// TIA Portal project "CalcOnSCADA_05" (V14)

(* hardware
DEVICE "S71500/ET200MP station_1"  S7-1500 station
   slot 0: "Rail_0"  Rack  6ES7 590-1***0-0AA0
   slot 1: "PLC_1"  CPU 1513-1 PN  6ES7 513-1AL01-0AB0  V2.1
      slot 3: "CPU display_1"  6ES7591-1AA00-0AA0
DEVICE "HMI_1"  TP900 Comfort
   slot 0: "TP900 Comfort"  TP900 Comfort  6AV2 124-0JC01-0AX0  14.0.1.0
   slot 1: "HMI_RT_1"  TP900 Comfort  6AV2 124-0JC01-0AX0  14.0.1.0
   slot 5: "HMI_1.IE_CP_1"  PROFINET Interface  14.0.1.0
      slot 1: "PROFINET Interface_1"  PROFINET Interface
         slot 1: "Port_1"  Port
         slot 2: "Port_2"  Port
   slot 7: "HMI_1.MPI/DP_CP_1"  MPI/DP Interface  14.0.1.0
*)

// ===== PLC "PLC_1"  CPU 1513-1 PN =====

VAR_GLOBAL   // PLC tag table "Default tag table"
   "positive" AT %M515.0 : Bool;
   "positiveOut" AT %M515.1 : Bool;
END_VAR

VAR_GLOBAL   // PLC tag table "Tag table_1"
   "Watchable" AT %M100.0 : LReal;
   "hjbhb" AT %M108.0 : LReal;
   "mb514" AT %MB514 : Byte;
END_VAR

TYPE "Digit"
   STRUCT
      visiComa : Bool;
      visiMinus : Bool;
      visible2 : Bool;
      visible3 : Bool;
      visible4 : Bool;
      visible5 : Bool;
      visible6 : Bool;
      visible7 : Bool;
      visible8 : Bool;
      visible9 : Bool;
      visible10 : Bool;
      visible11 : Bool;
      visible12 : Bool;
      visible13 : Bool;
      visible14 : Bool;
      visible15 : Bool;
      digit : Word;
   END_STRUCT;
END_TYPE

TYPE "Button"
   STRUCT
      b00 : Bool;
      b01 : Bool;
      b02 : Bool;
      b03 : Bool;
      b04 : Bool;
      b05 : Bool;
      click : Bool;
      oldClick : Bool;
   END_STRUCT;
END_TYPE

TYPE "Number"
   STRUCT
      coma : Bool;
      initOk : Bool;
      num2 : Bool;
      num3 : Bool;
      num4 : Bool;
      num5 : Bool;
      num6 : Bool;
      num7 : Bool;
      longI : LInt;
      I : Int;
      longTr : LReal;
      Tr : Real;
      longR : LReal;
      R : Real;
      pos : Int;   // Кількість десяткових розрядів
      posC : Int;   // Позиція коми
      posR : LInt;   // Вага десяткового розряду
   END_STRUCT;
END_TYPE

DATA_BLOCK "NUMs"   // DB1
{ S7_Optimized_Access := 'TRUE' }
VERSION : 0.1
   VAR
      Num : Array[0..31] of "Number";
      TEMP : Array[0..17] of LReal;
      TEMP2 : Array[0..17] of LInt;
      FaceLongI : String;
      FaceI : String;
      FaceLongR : String;
      FaceR : String;
      Index : Int;   // Індекс у масиві Num
      Action : Int;
      ActionBit : Bool;
      ActBit : Bool;   // Щоб виконати дію без =
      EquaBit : Bool;
      FaceLongFr : String;
      FaceFr : String;
      SizeI : Int;
      SizeAll : Int;
      Error : Bool;
      preError : Bool;
      TEN : Array[0..15] of LReal;
      bTEN : Array[0..15] of LReal;
   END_VAR
BEGIN
   bTEN[0] := 1.0E-15;
   bTEN[1] := 1.0E-14;
   bTEN[2] := 1.0E-13;
   bTEN[3] := 1.0E-12;
   bTEN[15] := 1.0;
   bTEN[9] := 1.0E-06;
   bTEN[10] := 1.0E-05;
   bTEN[11] := 0.0001;
   bTEN[12] := 0.001;
   bTEN[13] := 0.01;
   bTEN[14] := 0.1;
   bTEN[4] := 1.0E-11;
   bTEN[5] := 1.0E-10;
   bTEN[6] := 1.0E-09;
   bTEN[7] := 1.0E-08;
   bTEN[8] := 1.0E-07;
   TEN[0] := 1.0;
   TEN[1] := 10.0;
   TEN[2] := 100.0;
   TEN[3] := 1000.0;
   TEN[4] := 10000.0;
   TEN[5] := 100000.0;
   TEN[6] := 1000000.0;
   TEN[7] := 10000000.0;
   TEN[8] := 100000000.0;
   TEN[9] := 1000000000.0;
   TEN[10] := 10000000000.0;
   TEN[11] := 100000000000.0;
   TEN[12] := 1000000000000.0;
   TEN[13] := 10000000000000.0;
   TEN[14] := 100000000000000.0;
   TEN[15] := 1.0E+15;
END_DATA_BLOCK

// folder: Group_Misc

DATA_BLOCK "Digit_bl_10"   // DB10
{ S7_Optimized_Access := 'TRUE' }
VERSION : 0.1
   VAR
      Header : ArrayDBHeader;
      THIS : Array[0..15] of "Digit";
   END_VAR
BEGIN
   Header.LowerBound := 0;
   Header.UpperBound := 15;
   Header.Elements := 16;
   Header.PaddedSize := 18;
   Header.ElementSize := 18;
   THIS[0].digit := 16#1;
END_DATA_BLOCK

DATA_BLOCK "Butt_bl_200"   // DB200
{ S7_Optimized_Access := 'TRUE' }
VERSION : 0.1
   VAR
      Header : ArrayDBHeader;
      THIS : Array[0..31] of "Button";
   END_VAR
BEGIN
   Header.LowerBound := 0;
   Header.UpperBound := 31;
   Header.Elements := 32;
   Header.PaddedSize := 8;
   Header.ElementSize := 8;
END_DATA_BLOCK

// folder: System blocks/Program resources

DATA_BLOCK "DB_Timer_0"   // DB2
{ S7_Optimized_Access := 'TRUE' }
AUTHOR : Simatic
FAMILY : IEC
NAME : IEC_TMR
VERSION : 1.0
// stored: InstanceOfName IEC_TIMER
"IEC_TIMER"
BEGIN
END_DATA_BLOCK

// folder: (top level)

FUNCTION "Block_NumToD" : Void   // FC15, SCL
{ S7_Optimized_Access := 'TRUE' }
VERSION : 0.1
   VAR_INPUT
      inNumber : "Number";
   END_VAR
   VAR_TEMP
      tFaceLongR : String;
      tFaceLongI : String;
      tSizeAll : Int;
      tSizeFr : Int;
      ii : Int;
      i2 : Int;
      tShift : Word;
      tInt : Int;
      tShortStr : String;
      tDLongR : LReal;
      tLongR : LReal;
      tLongR2 : LReal;
      tLongI : LInt;
      tLongTr : LReal;
   END_VAR
   VAR CONSTANT
      word1 : Word := 16#1;
   END_VAR
BEGIN

   (*IF #inNumber.longI < 0 THEN
       #tAbsLongI := - #inNumber.longI; //знаходимо модуль
   ELSE
       #tAbsLongI := #inNumber.longI; //знаходимо модуль
   END_IF;
   #tAbsLongI := ABS(#inNumber.longI);*)

   #tFaceLongI      := S_CONV(#inNumber.longI);
   //"NUMs".FaceLongI := #tFaceLongI;
   "NUMs".FaceI     := S_CONV(#inNumber.I);
   #tFaceLongR      := S_CONV(#inNumber.longR);
   "NUMs".FaceLongR := #tFaceLongR;
   "NUMs".FaceR     := S_CONV(#inNumber.R);
   //"NUMs".FaceR := FC30(#tNumber.R);
   //"NUMs".FaceLongFr:= LREAL_TO_STRING(#inNumber.longTr);
   //"NUMs".FaceFr    := REAL_TO_STRING(#inNumber.Tr);

   #tLongR := ABS(#inNumber.longR);
   //#tLongR := ABS(#tLongR);
   #tLongI := ABS(#inNumber.longI);
   //#tLongI := ABS(#tLongI);
   #tLongTr := ABS(#inNumber.longTr);
   #tDLongR := #tLongR - #tLongTr;
   (*#tLongR := #inNumber.longR;
   #tLongI := #inNumber.longI;
   #tLongR := #tLongR * 10;
   #tLongI := LREAL_TO_LINT(#tLongR - 0.4999);
   #tDLongR := #tLongR - #tLongI;*)
   (*#i2 := 100;
   WHILE #ii <5 AND #i2 < 110 DO
       #ii += 1;
       #i2 += 1;
   END_WHILE;*)
   "NUMs".SizeI := LEN(#tFaceLongI); //намагаємося вирахувати кількість знакомісць до коми
   IF #tLongI < 1 THEN
       "NUMs".SizeI := 1;
   ELSE
       "NUMs".SizeI -= 1;
   END_IF;
   //"NUMs".TEMP[1]:=0;
   #tSizeFr := 0;    // 123456789012345
   WHILE #tDLongR > "NUMs".bTEN[#tSizeFr] AND #tSizeFr < (16-"NUMs".SizeI) DO
       "NUMs".TEMP[#tSizeFr] := #tDLongR;
       #tSizeFr += 1;
       //#tLongR := #tLongR * 10;
       #tLongR2 := "NUMs".TEN[#tSizeFr] * #tLongR ;
       //"NUMs".TEN[#tSizeFr] += 1;
       #tLongI := TRUNC(#tLongR2);
       "NUMs".TEMP2[#tSizeFr-1] := #tLongI;
       //#tInt := LREAL_TO_INT(#tLongR2 - 0.5);
       #tDLongR := #tLongR2 - LINT_TO_LREAL(#tLongI);  // +0.0000000000001;
       //#tDLongR := #tLongR2 - #tInt;
   END_WHILE;
   "NUMs".TEMP[#tSizeFr] := 88888888888888;
   "NUMs".TEMP2[#tSizeFr] := 88888888888888;

   #tFaceLongI := S_CONV(#tLongI);
   "NUMs".FaceLongI := #tFaceLongI;

   #tSizeAll := LEN(#tFaceLongI);
   "NUMs".SizeAll := #tSizeAll;
   "Block_CLS"();
   #tSizeAll := #tSizeAll - 1;
   (*
   #tShortStr := MID(IN := #tFaceLongI, L := 1, P := 2);
   #tInt := STRING_TO_INT(#tShortStr);
   #tShift := SHL(IN := #word1, N := #tInt);
   "Digit_bl_10"."THIS"[0].digit := #tShift;
   *)
   FOR #ii := 1 TO #tSizeAll DO
       #tShift := SHL(IN := #word1, N := S_CONV(MID(IN := #tFaceLongI, L := 1, P := #ii + 1)));
       "Digit_bl_10".THIS[#tSizeAll - #ii].digit := #tShift;
   END_FOR;
   IF #tSizeFr > 0 THEN
       "Digit_bl_10".THIS[#tSizeFr].visiComa := TRUE;
   END_IF;

   #ii := #tSizeFr;
   IF #tSizeAll>#tSizeFr THEN
       #inNumber.pos := #tSizeAll - 1;     //задля "Block_setMinus"
   ELSE
       #inNumber.pos := #tSizeFr;     //задля "Block_setMinus"
       REPEAT
           "Digit_bl_10".THIS[#ii].digit := 1;
           #ii -= 1;
       UNTIL (#ii-#tSizeAll)<0
       END_REPEAT;
   END_IF;

   "Block_setMinus"();
END_FUNCTION

FUNCTION "Block_100" : Void   // FC100, SCL
{ S7_Optimized_Access := 'TRUE' }
VERSION : 0.1
   VAR_TEMP
      ii : Int;
      tpos : Int;
      tButton : "Button";
      tLReal : LReal;
      tLInt : LInt;
   END_VAR
BEGIN


   //      =
   #tButton := "Butt_bl_200".THIS[24];
   IF (#tButton.click <> #tButton.oldClick) AND NOT "NUMs".Error THEN
       "Block_Equal"();
   END_IF;
   //      /
   #tButton := "Butt_bl_200".THIS[20];
   IF #tButton.click <> #tButton.oldClick THEN
       "Block_Action"();
       "NUMs".Action := 4;
   END_IF;
   //      *
   #tButton := "Butt_bl_200".THIS[21];
   IF #tButton.click <> #tButton.oldClick THEN
       "Block_Action"();
       "NUMs".Action := 3;
   END_IF;
   //      -
   #tButton := "Butt_bl_200".THIS[22];
   IF #tButton.click <> #tButton.oldClick THEN
       "Block_Action"();
       "NUMs".Action := 2;
   END_IF;
   //      +
   #tButton := "Butt_bl_200".THIS[23];
   IF #tButton.click <> #tButton.oldClick THEN
       "Block_Action"();
       "NUMs".Action := 1;
   END_IF;

   //      Coma
   #tButton := "Butt_bl_200".THIS[12];
   IF #tButton.click <> #tButton.oldClick THEN
       "NUMs".Num["NUMs".Index].initOk := true;
       IF "NUMs".Num["NUMs".Index].coma THEN
           ;
       ELSE
           "Digit_bl_10".THIS[0].visiComa := true;
       END_IF;
       "NUMs".Num["NUMs".Index].coma := true;
   END_IF;
   //      CE
   #tButton := "Butt_bl_200".THIS[17];
   IF #tButton.click <> #tButton.oldClick THEN
       "Block_CE"();
   END_IF;
   //      C
   #tButton := "Butt_bl_200".THIS[18];
   IF #tButton.click <> #tButton.oldClick THEN
       "Block_C"();
   END_IF;
   //      0
   #tButton := "Butt_bl_200".THIS[10];
   IF #tButton.click <> #tButton.oldClick AND ("NUMs".Num["NUMs".Index].pos < 15) THEN
       "Block_num Butt" ( iInt:=0, iDigit:=1 );
   END_IF;
   //      1
   #tButton := "Butt_bl_200".THIS[1];
   IF #tButton.click <> #tButton.oldClick AND ("NUMs".Num["NUMs".Index].pos < 15) THEN
       "Block_num Butt" ( iInt:=1, iDigit:=2 );
   END_IF;
   //      2
   #tButton := "Butt_bl_200".THIS[2];
   IF #tButton.click <> #tButton.oldClick AND ("NUMs".Num["NUMs".Index].pos < 15) THEN
       "Block_num Butt" ( iInt:=2, iDigit:=4 );
   END_IF;
   //      3
   #tButton := "Butt_bl_200".THIS[3];
   IF #tButton.click <> #tButton.oldClick AND ("NUMs".Num["NUMs".Index].pos < 15) THEN
       "Block_num Butt" ( iInt:=3, iDigit:=8 );
   END_IF;
   //      4
   #tButton := "Butt_bl_200".THIS[4];
   IF #tButton.click <> #tButton.oldClick AND ("NUMs".Num["NUMs".Index].pos < 15) THEN
       "Block_num Butt"(iInt := 4, iDigit := 16);
   END_IF;
   //      5
   #tButton := "Butt_bl_200".THIS[5];
   IF #tButton.click <> #tButton.oldClick AND ("NUMs".Num["NUMs".Index].pos < 15) THEN
       "Block_num Butt" ( iInt:=5, iDigit:=32 );
   END_IF;
   //      6
   #tButton := "Butt_bl_200".THIS[6];
   IF #tButton.click <> #tButton.oldClick AND ("NUMs".Num["NUMs".Index].pos < 15) THEN
       "Block_num Butt" ( iInt:=6, iDigit:=64 );
   END_IF;
   //      7
   #tButton := "Butt_bl_200".THIS[7];
   IF #tButton.click <> #tButton.oldClick AND ("NUMs".Num["NUMs".Index].pos < 15) THEN
       "Block_num Butt" ( iInt:=7, iDigit:=128 );
   END_IF;
   //      8
   #tButton := "Butt_bl_200".THIS[8];
   IF #tButton.click <> #tButton.oldClick AND ("NUMs".Num["NUMs".Index].pos < 15) THEN
       "Block_num Butt"(iInt := 8, iDigit := 256);
   END_IF;
   //      9
   #tButton := "Butt_bl_200".THIS[9];
   IF #tButton.click <> #tButton.oldClick AND ("NUMs".Num["NUMs".Index].pos < 15) THEN
       "Block_num Butt" ( iInt:=9, iDigit:=512 );
   END_IF;

   //      +-
   #tButton := "Butt_bl_200".THIS[11];
   IF (#tButton.click <> #tButton.oldClick) AND NOT "NUMs".Error THEN
       "Block_Minus"();
   END_IF;
END_FUNCTION

ORGANIZATION_BLOCK "Main"   // OB1, STL, ProgramCycle
TITLE = "Main Program Sweep (Cycle)"
{ S7_Optimized_Access := 'TRUE' }
VERSION : 0.1
   VAR_INPUT
      Initial_Call : Bool;   // Initial call of this OB
      Remanence : Bool;   // =True, if remanent data are available
   END_VAR
BEGIN

REGION Network 1
         CALL  "Block_100";
END_REGION

REGION Network 2
         CALL  "Block_200";
END_REGION

REGION Network 3
         CALL  "Block_99";
END_REGION
END_ORGANIZATION_BLOCK

ORGANIZATION_BLOCK "Programming error"   // OB121, LAD, ProgrammingError
{ S7_Optimized_Access := 'TRUE' }
VERSION : 0.1
   VAR_INPUT
      BlockNr : UInt;   // Number of causing block
      Reaction : USInt;   // 0:ignore, 1:substitute, 2:skip
      Fault_ID : Byte;   // Fault identifier
      BlockType : USInt;   // 16#01:OB, 16#02:FC, 16#03:FB, 16#04:SFC, 16#05:SFB, 16#06:DB: Type of block causing the error
      Area : USInt;   // Area where the error occured
      DBNr : DB_ANY;   // DB number if Area = DB or DI
      Csg_OBNr : OB_Any;   // Number of OB causing the error
      Csg_Prio : USInt;   // Priority of OB causing the error
      Width : USInt;   // 0:bit, 1:byte, 2:word, 3:dword, 4:lword
   END_VAR
BEGIN

REGION Network 1
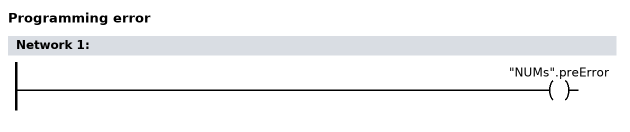
   RUNG wire#powerrail
      Coil( "NUMs".preError )
   END_RUNG
   // the same network as SCL:
   "NUMs".preError := TRUE;
END_REGION
END_ORGANIZATION_BLOCK

// folder: Group_100

FUNCTION "Block_CLS" : Void   // FC2, SCL
{ S7_Optimized_Access := 'TRUE' }
VERSION : 0.1
   VAR_TEMP
      ii : Int;
   END_VAR
BEGIN


   FOR #ii := 0 TO 15 DO
       "Digit_bl_10".THIS[#ii].digit := 0;
   END_FOR;
   "Block_unComa"();   //прибираю коми
   "Block_unMinus"();  //прибираю мінуси
END_FUNCTION

FUNCTION "Block_num Butt" : Void   // FC11, SCL
{ S7_Optimized_Access := 'TRUE' }
VERSION : 0.1
   VAR_INPUT
      iDigit : Word;
      iInt : Int;
   END_VAR
   VAR_TEMP
      tpos : Int;
      tLReal : LReal;
   END_VAR
BEGIN

   IF "NUMs".Error THEN
       "Block_C"();
   END_IF;

   IF "NUMs".ActionBit THEN
       "Block_CE"();
       "NUMs".ActionBit := false;
   END_IF;

   IF "NUMs".EquaBit THEN
       "Block_CE"();
       "NUMs".EquaBit := false;
   END_IF;

   IF "NUMs".Num["NUMs".Index].initOk THEN
       "NUMs".Num["NUMs".Index].pos += 1;
       #tpos := "NUMs".Num["NUMs".Index].pos;
       WHILE #tpos > 0 DO
           "Digit_bl_10".THIS[#tpos].digit :=
           "Digit_bl_10".THIS[#tpos - 1].digit;
           #tpos -= 1;
       END_WHILE;
       IF "NUMs".Num["NUMs".Index].coma THEN
           "NUMs".Num["NUMs".Index].posR *=10;
           #tLReal := #iInt;
           "NUMs".Num["NUMs".Index].longR :=
           #tLReal / "NUMs".Num["NUMs".Index].posR + "NUMs".Num["NUMs".Index].longR;
           "NUMs".Num["NUMs".Index].R := "NUMs".Num["NUMs".Index].longR;   //звичайний ріел
           (*        
           "NUMs".Num["NUMs".Index].longFr :=
           "NUMs".Num["NUMs".Index].longR - "NUMs".Num["NUMs".Index].longI;
           *)
           "NUMs".Num["NUMs".Index].longTr :=
           #tLReal / "NUMs".Num["NUMs".Index].posR + "NUMs".Num["NUMs".Index].longTr;
           "NUMs".Num["NUMs".Index].Tr := "NUMs".Num["NUMs".Index].longTr;
       ELSE
           "NUMs".Num["NUMs".Index].longI := 10 * "NUMs".Num["NUMs".Index].longI + #iInt;
           "NUMs".Num["NUMs".Index].I := 10 * "NUMs".Num["NUMs".Index].I + #iInt;
           "NUMs".Num["NUMs".Index].longR := 10 * "NUMs".Num["NUMs".Index].longR + #iInt;
           "NUMs".Num["NUMs".Index].R := "NUMs".Num["NUMs".Index].longR;   //звичайний ріел
       END_IF;
   ELSE
       "NUMs".Num["NUMs".Index].longI := #iInt;
       "NUMs".Num["NUMs".Index].I := #iInt;
       "NUMs".Num["NUMs".Index].longR := #iInt;
       "NUMs".Num["NUMs".Index].R := #iInt;
   END_IF;

   "Digit_bl_10".THIS[0].digit := #iDigit; //

   IF "NUMs".Num["NUMs".Index].coma THEN
       "NUMs".Num["NUMs".Index].posC +=1;
       "Block_unComa"();//прибираю коми
       "Digit_bl_10".THIS["NUMs".Num["NUMs".Index].posC].visiComa := true;   //
   END_IF;
   "Block_setMinus"();

   IF #iInt = 0 THEN
       ;
   ELSE
       "NUMs".Num["NUMs".Index].initOk := true;
   END_IF;
END_FUNCTION

FUNCTION "Block_Equal" : Void   // FC12, SCL
{ S7_Optimized_Access := 'TRUE' }
VERSION : 0.1
   VAR_TEMP
      tLReal : LReal;
      tButton : "Button";
      tLInt : LInt;
   END_VAR
BEGIN

       "NUMs".Index := 0;
       #tLReal := "NUMs".Num[0].longR;
       CASE "NUMs".Action OF
           1:
               "NUMs".Num[0].longR := #tLReal + "NUMs".Num[1].longR;
           2:
               "NUMs".Num[0].longR := #tLReal - "NUMs".Num[1].longR;
           3:
               "NUMs".Num[0].longR := #tLReal * "NUMs".Num[1].longR;
           4:
               "NUMs".Num[0].longR := #tLReal / "NUMs".Num[1].longR;
       END_CASE;

   "Block_ActCase"();
   "Block_NumToD"("NUMs".Num[0]);

   "NUMs".EquaBit := TRUE;
   "NUMs".ActBit := FALSE;
END_FUNCTION

FUNCTION "Block_unComa" : Void   // FC13, SCL
{ S7_Optimized_Access := 'TRUE' }
VERSION : 0.1
   VAR_TEMP
      ii : Int;
   END_VAR
BEGIN

   FOR #ii := 0 TO 15 DO
       "Digit_bl_10".THIS[#ii].visiComa := FALSE;
   END_FOR;
END_FUNCTION

FUNCTION "Block_CE" : Void   // FC14, SCL
{ S7_Optimized_Access := 'TRUE' }
VERSION : 0.1
   VAR_TEMP
      ii : Int;
   END_VAR
BEGIN

   "Block_NumCE"("NUMs".Index);
END_FUNCTION

FUNCTION "Block_Zeroing" : Void   // FC16, SCL
{ S7_Optimized_Access := 'TRUE' }
VERSION : 0.1
   VAR_INPUT
      iIndex : Int;
   END_VAR
BEGIN


   "NUMs".Num[#iIndex].longI := 0;
   "NUMs".Num[#iIndex].I := 0;
   "NUMs".Num[#iIndex].longR := 0.0;
   "NUMs".Num[#iIndex].R := 0.0;
   "NUMs".Num[#iIndex].longTr := 0.0;
   "NUMs".Num[#iIndex].Tr := 0.0;
END_FUNCTION

FUNCTION "Block_C" : Void   // FC17, SCL
{ S7_Optimized_Access := 'TRUE' }
VERSION : 0.1
BEGIN

   "NUMs".ActionBit := FALSE;
   "NUMs".ActBit := FALSE;
   "NUMs".Action := 0;
   "NUMs".Index := 0;
   "Block_NumCE"(0);
   "Block_NumCE"(1);

   "NUMs".Error := FALSE;
   "NUMs".preError := FALSE;
END_FUNCTION

FUNCTION "Block_NumCE" : Void   // FC18, SCL
{ S7_Optimized_Access := 'TRUE' }
VERSION : 0.1
   VAR_INPUT
      iIndex : Int;
   END_VAR
BEGIN

   "NUMs".Num[#iIndex].initOk := false;
   "NUMs".Num[#iIndex].coma := false;
   "NUMs".Num[#iIndex].pos := 0;
   "NUMs".Num[#iIndex].posC := 0;
   "NUMs".Num[#iIndex].posR := 1;

   "Block_Zeroing"(#iIndex);
   "Block_CLS"();

   //"Digit_bl_10"."THIS"[0].visible0 := false;
   "Digit_bl_10".THIS[0].digit := 1;
END_FUNCTION

FUNCTION "Block_LAD" : Void   // FC19, LAD
{ S7_Optimized_Access := 'TRUE' }
VERSION : 0.1
BEGIN
END_FUNCTION

FUNCTION "Block_Action" : Void   // FC20, SCL
{ S7_Optimized_Access := 'TRUE' }
VERSION : 0.1
BEGIN

   IF "NUMs".ActBit AND (NOT "NUMs".ActionBit) THEN
       "Block_Equal"();
   END_IF;
   "NUMs".ActBit := TRUE;

   "NUMs".Index := 1;
   "NUMs".ActionBit := TRUE;
END_FUNCTION

FUNCTION "Block_ActCase" : Void   // FC21, SCL
{ S7_Optimized_Access := 'TRUE' }
VERSION : 0.1
BEGIN

   "NUMs".Num[0].R := "NUMs".Num[0].longR;
   (*"NUMs".Num[0].longFr := FRAC_LREAL("NUMs".Num[0].longR);
   "NUMs".Num[0].Fr := "NUMs".Num[0].longFr;*)

   //"NUMs".Num[0].longI := LREAL_TO_LINT("NUMs".Num[0].longR - 0.499999);
   "NUMs".Num[0].longI := TRUNC("NUMs".Num[0].longR);
   "NUMs".Num[0].I     := TRUNC("NUMs".Num[0].longR);

   "NUMs".Num[0].longTr := TRUNC("NUMs".Num[0].longR);
   "NUMs".Num[0].Tr     := TRUNC("NUMs".Num[0].longR);
END_FUNCTION

FUNCTION "Block_setMinus" : Void   // FC22, SCL
{ S7_Optimized_Access := 'TRUE' }
VERSION : 0.1
BEGIN


   IF "NUMs".Num["NUMs".Index].longR < 0 THEN
       "Block_unMinus"();  //прибираю мінуси
       "Digit_bl_10".THIS["NUMs".Num["NUMs".Index].pos].visiMinus := TRUE;        //
   END_IF;
END_FUNCTION

FUNCTION "Block_unMinus" : Void   // FC23, SCL
{ S7_Optimized_Access := 'TRUE' }
VERSION : 0.1
   VAR_TEMP
      ii : Int;
   END_VAR
BEGIN

   FOR #ii := 0 TO 15 DO
       "Digit_bl_10".THIS[#ii].visiMinus := FALSE;
   END_FOR;
END_FUNCTION

FUNCTION "Block_Minus" : Void   // FC101, SCL
{ S7_Optimized_Access := 'TRUE' }
VERSION : 0.1
BEGIN

   //"mb514" := "mb514" + 1;
   //invert
   "Digit_bl_10".THIS["NUMs".Num["NUMs".Index].pos].visiMinus := NOT "Digit_bl_10".THIS["NUMs".Num["NUMs".Index].pos].visiMinus;
   "NUMs".Num["NUMs".Index].longR := -"NUMs".Num["NUMs".Index].longR;



   //
END_FUNCTION

// folder: Group_200

FUNCTION "Block_200" : Void   // FC200, FBD
{ S7_Optimized_Access := 'TRUE' }
VERSION : 0.1
BEGIN

REGION Network 1
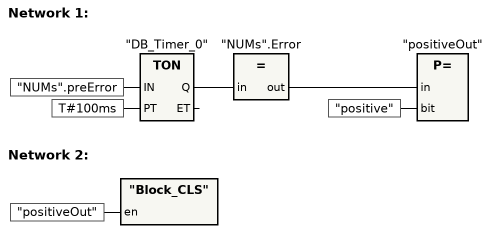
   "DB_Timer_0".TON(IN := "NUMs".preError, PT := T#100ms);
   "NUMs".Error := "DB_Timer_0".Q;
   "positiveOut" := "DB_Timer_0".Q AND NOT "positive";   // rising edge
   "positive" := "DB_Timer_0".Q;
END_REGION

REGION Network 2
   IF "positiveOut" THEN "Block_CLS"(); END_IF;
END_REGION
END_FUNCTION

// folder: Group_Misc

FUNCTION "Block_Start" : Void   // FC1, SCL
{ S7_Optimized_Access := 'TRUE' }
VERSION : 0.1
BEGIN

   //"Watchable" := 5.6;
END_FUNCTION

FUNCTION "Block_99" : Void   // FC99, SCL
{ S7_Optimized_Access := 'TRUE' }
VERSION : 0.1
   VAR_TEMP
      ii : Int;
   END_VAR
BEGIN

   FOR #ii := 0 TO 31 DO
       "Butt_bl_200".THIS[#ii].oldClick := "Butt_bl_200".THIS[#ii].click;
   END_FOR;
END_FUNCTION

ORGANIZATION_BLOCK "Startup"   // OB100, STL, Startup
TITLE = "Complete Restart"
{ S7_Optimized_Access := 'TRUE' }
VERSION : 0.1
   VAR_INPUT
      LostRetentive : Bool;   // True if retentive data are lost
      LostRTC : Bool;   // True if date and time are lost
   END_VAR
BEGIN

REGION Network 1
   //CALL  "Block_FCstart"
END_REGION
END_ORGANIZATION_BLOCK

(* ===== HMI "HMI_RT_1" =====
system functions are stored by id; their names below are inferred from use
connection "HMI_Connection_1": ETHERNET, S7_1500_OMS

HMI tags "Default tag table"
   "Tag_ScreenNumber" : UInt, internal
   "Watchable" : LReal = PLC Watchable AT %M100.0, 1 s
   "Digit_bl_10_THIS{0}_visible0" : Bool = PLC Digit_bl_10.THIS[0].visiComa, 1 s
   "Digit_bl_10_THIS{0}_digarray{0}" : Word = PLC Digit_bl_10.THIS[0].digit, 1 s
   "Digit_bl_10_THIS[1]_digarray[0]" : Word = PLC Digit_bl_10.THIS[1].digit AT %DB1.DBX0.0, 1 s
   "Digit_bl_10_THIS[2]_digarray[0]" : Word = PLC Butt_bl_200.THIS[5].click AT %DB1.DBX0.0, 1 s
   "Digit_bl_10_THIS[3]_digarray[0]" : Word = PLC Butt_bl_200.THIS[12].click AT %DB1.DBX0.0, 1 s
   "Digit_bl_10_THIS[4]_digarray[0]" : Word = PLC Butt_bl_200.THIS[4].click AT %DB1.DBX0.0, 1 s
   "Digit_bl_10_THIS[5]_digarray[0]" : Word = PLC Butt_bl_200.THIS[3].click AT %DB1.DBX0.0, 1 s
   "Digit_bl_10_THIS[6]_digarray[0]" : Word = PLC Digit_bl_10.THIS[6].digit AT %DB1.DBX0.0, 1 s
   "Digit_bl_10_THIS[7]_digarray[0]" : Word = PLC Digit_bl_10.THIS[7].digit AT %DB1.DBX0.0, 1 s
   "Digit_bl_10_THIS[8]_digarray[0]" : Word = PLC Butt_bl_200.THIS[7].click AT %DB1.DBX0.0, 1 s
   "Digit_bl_10_THIS[9]_digarray[0]" : Word = PLC Butt_bl_200.THIS[2].click AT %DB1.DBX0.0, 1 s
   "Digit_bl_10_THIS[10]_digarray[0]" : Word = PLC Butt_bl_200.THIS[1].click AT %DB1.DBX0.0, 1 s
   "Digit_bl_10_THIS[11]_digarray[0]" : Word = PLC Digit_bl_10.THIS[11].digit AT %DB1.DBX0.0, 1 s
   "Digit_bl_10_THIS[12]_digarray[0]" : Word = PLC Digit_bl_10.THIS[12].digit AT %DB1.DBX0.0, 1 s
   "Digit_bl_10_THIS[13]_digarray[0]" : Word = PLC Digit_bl_10.THIS[13].digit AT %DB1.DBX0.0, 1 s
   "Digit_bl_10_THIS[14]_digarray[0]" : Word = PLC Digit_bl_10.THIS[14].digit AT %DB1.DBX0.0, 1 s
   "Digit_bl_10_THIS[15]_digarray[0]" : Word = PLC Butt_bl_200.THIS[6].click AT %DB1.DBX0.0, 1 s
   "Digit_bl_10_THIS{15}_visible0" : Bool = PLC Digit_bl_10.THIS[15].visiComa, 1 s
   "Digit_bl_10_THIS{1}_visible0" : Bool = PLC Digit_bl_10.THIS[1].visiComa, 1 s
   "Digit_bl_10_THIS{2}_visible0" : Bool = PLC Digit_bl_10.THIS[2].visiComa, 1 s
   "Digit_bl_10_THIS{3}_visible0" : Bool = PLC Digit_bl_10.THIS[3].visiComa, 1 s
   "Digit_bl_10_THIS{4}_visible0" : Bool = PLC Digit_bl_10.THIS[4].visiComa, 1 s
   "Digit_bl_10_THIS{5}_visible0" : Bool = PLC Digit_bl_10.THIS[5].visiComa, 1 s
   "Digit_bl_10_THIS{6}_visible0" : Bool = PLC Digit_bl_10.THIS[6].visiComa, 1 s
   "Digit_bl_10_THIS{7}_visible0" : Bool = PLC Digit_bl_10.THIS[7].visiComa, 1 s
   "Digit_bl_10_THIS{8}_visible0" : Bool = PLC Digit_bl_10.THIS[8].visiComa, 1 s
   "Digit_bl_10_THIS{9}_visible0" : Bool = PLC Digit_bl_10.THIS[9].visiComa, 1 s
   "Digit_bl_10_THIS{10}_visible0" : Bool = PLC Digit_bl_10.THIS[10].visiComa, 1 s
   "Digit_bl_10_THIS{11}_visible0" : Bool = PLC Digit_bl_10.THIS[11].visiComa, 1 s
   "Digit_bl_10_THIS{12}_visible0" : Bool = PLC Digit_bl_10.THIS[12].visiComa, 1 s
   "Digit_bl_10_THIS{13}_visible0" : Bool = PLC Digit_bl_10.THIS[13].visiComa, 1 s
   "Digit_bl_10_THIS{14}_visible0" : Bool = PLC Digit_bl_10.THIS[14].visiComa, 1 s
   "NUMs_Error" : Bool = PLC NUMs.Error, 1 s
   "Digit_bl_10_THIS{0}_visiMinus" : Bool = PLC Butt_bl_200.THIS[17].click, 1 s
   "Digit_bl_10_THIS{1}_visiMinus" : Bool = PLC Digit_bl_10.THIS[1].visiMinus, 1 s
   "Digit_bl_10_THIS{2}_visiMinus" : Bool = PLC Digit_bl_10.THIS[2].visiMinus, 1 s
   "Digit_bl_10_THIS{3}_visiMinus" : Bool = PLC Digit_bl_10.THIS[3].visiMinus, 1 s
   "Digit_bl_10_THIS{4}_visiMinus" : Bool = PLC Digit_bl_10.THIS[4].visiMinus, 1 s
   "Digit_bl_10_THIS{5}_visiMinus" : Bool = PLC Digit_bl_10.THIS[5].visiMinus, 1 s
   "Digit_bl_10_THIS{6}_visiMinus" : Bool = PLC Digit_bl_10.THIS[6].visiMinus, 1 s
   "Digit_bl_10_THIS{7}_visiMinus" : Bool = PLC Digit_bl_10.THIS[7].visiMinus, 1 s
   "Digit_bl_10_THIS{8}_visiMinus" : Bool = PLC Digit_bl_10.THIS[8].visiMinus, 1 s
   "Digit_bl_10_THIS{9}_visiMinus" : Bool = PLC Digit_bl_10.THIS[9].visiMinus, 1 s
   "Digit_bl_10_THIS{10}_visiMinus" : Bool = PLC Digit_bl_10.THIS[10].visiMinus, 1 s
   "Digit_bl_10_THIS{11}_visiMinus" : Bool = PLC Digit_bl_10.THIS[11].visiMinus, 1 s
   "Digit_bl_10_THIS{12}_visiMinus" : Bool = PLC Digit_bl_10.THIS[12].visiMinus, 1 s
   "Digit_bl_10_THIS{13}_visiMinus" : Bool = PLC Digit_bl_10.THIS[13].visiMinus, 1 s
   "Digit_bl_10_THIS{14}_visiMinus" : Bool = PLC Digit_bl_10.THIS[14].visiMinus, 1 s
   "Digit_bl_10_THIS{15}_visiMinus" : Bool = PLC Digit_bl_10.THIS[15].visiMinus, 1 s

HMI tags "HMI table Click"
   "Butt_bl_200_THIS{1}_click" : Bool = PLC Butt_bl_200.THIS[1].click, 100 ms
   "Butt_bl_200_THIS{10}_click" : Bool = PLC Butt_bl_200.THIS[10].click, 100 ms
   "Butt_bl_200_THIS{11}_click" : Bool = PLC Butt_bl_200.THIS[11].click, 100 ms
   "Butt_bl_200_THIS{12}_click" : Bool = PLC Butt_bl_200.THIS[12].click, 100 ms
   "Butt_bl_200_THIS{13}_click" : Bool = PLC Butt_bl_200.THIS[13].click, 1 s
   "Butt_bl_200_THIS{14}_click" : Bool = PLC Butt_bl_200.THIS[14].click, 1 s
   "Butt_bl_200_THIS{15}_click" : Bool = PLC Butt_bl_200.THIS[15].click, 1 s
   "Butt_bl_200_THIS{16}_click" : Bool = PLC Butt_bl_200.THIS[16].click, 1 s
   "Butt_bl_200_THIS{17}_click" : Bool = PLC Butt_bl_200.THIS[17].click, 1 s
   "Butt_bl_200_THIS{18}_click" : Bool = PLC Butt_bl_200.THIS[18].click, 1 s
   "Butt_bl_200_THIS{2}_click" : Bool = PLC Butt_bl_200.THIS[2].click, 100 ms
   "Butt_bl_200_THIS{3}_click" : Bool = PLC Butt_bl_200.THIS[3].click, 100 ms
   "Butt_bl_200_THIS{4}_click" : Bool = PLC Butt_bl_200.THIS[4].click, 100 ms
   "Butt_bl_200_THIS{5}_click" : Bool = PLC Butt_bl_200.THIS[5].click, 100 ms
   "Butt_bl_200_THIS{6}_click" : Bool = PLC Butt_bl_200.THIS[6].click, 100 ms
   "Butt_bl_200_THIS{7}_click" : Bool = PLC Butt_bl_200.THIS[7].click, 100 ms
   "Butt_bl_200_THIS{8}_click" : Bool = PLC Butt_bl_200.THIS[8].click, 100 ms
   "Butt_bl_200_THIS{9}_click" : Bool = PLC Butt_bl_200.THIS[9].click, 100 ms
   "Butt_bl_200_THIS{19}_click" : Bool = PLC Butt_bl_200.THIS[19].click AT %DB1.DBX0.0, 1 s
   "Butt_bl_200_THIS{20}_click" : Bool = PLC Butt_bl_200.THIS[20].click AT %DB1.DBX0.0, 1 s
   "Butt_bl_200_THIS{21}_click" : Bool = PLC Butt_bl_200.THIS[21].click AT %DB1.DBX0.0, 1 s
   "Butt_bl_200_THIS{22}_click" : Bool = PLC Butt_bl_200.THIS[22].click AT %DB1.DBX0.0, 1 s
   "Butt_bl_200_THIS{23}_click" : Bool = PLC Butt_bl_200.THIS[23].click AT %DB1.DBX0.0, 1 s
   "Butt_bl_200_THIS{24}_click" : Bool = PLC Butt_bl_200.THIS[24].click AT %DB1.DBX0.0, 1 s

screen "Root screen" 800x420, template "Template_1"
   on GenerateScreen: SetTag("Tag_ScreenNumber", 1)
   IOField "I/O field_1" at 105,99 size 400x40; FormatPattern 9
      ProcessValue <- "Watchable"
   Button "Button_1" at 105,250 size 102x42; TextOff '1'
      on Press: InvertBit("Butt_bl_200_THIS{1}_click")
   Button "Button_2" at 204,250 size 102x42; TextOff '2'
      on Press: InvertBit("Butt_bl_200_THIS{2}_click")
   Button "Button_3" at 304,250 size 102x42; TextOff '3'
      on Press: InvertBit("Butt_bl_200_THIS{3}_click")
   Button "Button_4" at 105,210 size 102x42; TextOff '4'
      on Press: InvertBit("Butt_bl_200_THIS{4}_click")
   Button "Button_5" at 205,210 size 102x42; TextOff '5'
      on Press: InvertBit("Butt_bl_200_THIS{5}_click")
   Button "Button_6" at 305,210 size 102x42; TextOff '6'
      on Press: InvertBit("Butt_bl_200_THIS{6}_click")
   Button "Button_7" at 105,170 size 102x42; TextOff '7'
      on Press: InvertBit("Butt_bl_200_THIS{7}_click")
   Button "Button_8" at 205,170 size 102x42; TextOff '8'
      on Press: InvertBit("Butt_bl_200_THIS{8}_click")
   Button "Button_9" at 305,170 size 102x42; TextOff '9'
      on Press: InvertBit("Butt_bl_200_THIS{9}_click")
   Button "Button_10" at 205,290 size 102x42; TextOff '0'
      on Press: InvertBit("Butt_bl_200_THIS{10}_click")
   Button "Button_11" at 105,290 size 102x42; TextOff '±'
      on Click: InvertBit("Butt_bl_200_THIS{11}_click")
   Button "Button_12" at 305,290 size 102x42; TextOff ','
      on Click: InvertBit("Butt_bl_200_THIS{12}_click")
   Button "Button_13" at 105,90 size 102x42; TextOff ','
   Button "Button_14" at 205,90 size 102x42; TextOff ','
   Button "Button_15" at 305,90 size 102x42; TextOff ','
   Button "Button_16" at 405,90 size 102x42; TextOff ','
   Button "Button_17" at 105,130 size 102x42; TextOff 'CE'
      on Click: InvertBit("Butt_bl_200_THIS{17}_click")
   Button "Button_18" at 205,130 size 102x42; TextOff 'C'
      on Click: InvertBit("Butt_bl_200_THIS{18}_click")
   Button "Button_19" at 305,130 size 102x42; TextOff ','
   Button "Button_20" at 405,130 size 102x42; TextOff '÷'
      on Click: InvertBit("Butt_bl_200_THIS{20}_click")
   Button "Button_21" at 405,170 size 102x42; TextOff '×'
      on Click: InvertBit("Butt_bl_200_THIS{21}_click")
   Button "Button_22" at 405,210 size 102x42; TextOff '–'
      on Click: InvertBit("Butt_bl_200_THIS{22}_click")
   Button "Button_23" at 405,250 size 102x42; TextOff '+'
      on Click: InvertBit("Butt_bl_200_THIS{23}_click")
   Button "Button_24" at 405,290 size 102x42; TextOff '='
      on Click: InvertBit("Butt_bl_200_THIS{24}_click")
   TextField "Text_dot" at 498,52 size 20x30; Text ','
      Visibility <- "Digit_bl_10_THIS{0}_visible0"
   TextField "Text field_0" at 480,40 size 30x50; Text '0'
      Visibility <- "Digit_bl_10_THIS{0}_digarray{0}"
   TextField "Text field_1" at 480,40 size 30x50; Text '1'
      Visibility <- "Digit_bl_10_THIS{0}_digarray{0}"
   TextField "Text field_2" at 480,40 size 30x50; Text '2'
      Visibility <- "Digit_bl_10_THIS{0}_digarray{0}"
   TextField "Text field_3" at 480,40 size 30x50; Text '3'
      Visibility <- "Digit_bl_10_THIS{0}_digarray{0}"
   TextField "Text field_4" at 480,40 size 30x50; Text '4'
      Visibility <- "Digit_bl_10_THIS{0}_digarray{0}"
   TextField "Text field_5" at 480,40 size 30x50; Text '5'
      Visibility <- "Digit_bl_10_THIS{0}_digarray{0}"
   TextField "Text field_6" at 480,40 size 30x50; Text '6'
      Visibility <- "Digit_bl_10_THIS{0}_digarray{0}"
   TextField "Text field_7" at 480,40 size 30x50; Text '7'
      Visibility <- "Digit_bl_10_THIS{0}_digarray{0}"
   TextField "Text field_8" at 480,40 size 30x50; Text '8'
      Visibility <- "Digit_bl_10_THIS{0}_digarray{0}"
   TextField "Text field_9" at 480,40 size 30x50; Text '9'
      Visibility <- "Digit_bl_10_THIS{0}_digarray{0}"
   Group "Group_0" at 480,40 size 38x50
   TextField "Text_dot_1" at 473,52 size 20x30; Text ','
      Visibility <- "Digit_bl_10_THIS{1}_visible0"
   TextField "Text field_10" at 455,40 size 30x50; Text '0'
      Visibility <- "Digit_bl_10_THIS[1]_digarray[0]"
   TextField "Text field_11" at 455,40 size 30x50; Text '1'
      Visibility <- "Digit_bl_10_THIS[1]_digarray[0]"
   TextField "Text field_12" at 455,40 size 30x50; Text '2'
      Visibility <- "Digit_bl_10_THIS[1]_digarray[0]"
   TextField "Text field_13" at 455,40 size 30x50; Text '3'
      Visibility <- "Digit_bl_10_THIS[1]_digarray[0]"
   TextField "Text field_14" at 455,40 size 30x50; Text '4'
      Visibility <- "Digit_bl_10_THIS[1]_digarray[0]"
   TextField "Text field_15" at 455,40 size 30x50; Text '5'
      Visibility <- "Digit_bl_10_THIS[1]_digarray[0]"
   TextField "Text field_16" at 455,40 size 30x50; Text '6'
      Visibility <- "Digit_bl_10_THIS[1]_digarray[0]"
   TextField "Text field_17" at 455,40 size 30x50; Text '7'
      Visibility <- "Digit_bl_10_THIS[1]_digarray[0]"
   TextField "Text field_18" at 455,40 size 30x50; Text '8'
      Visibility <- "Digit_bl_10_THIS[1]_digarray[0]"
   TextField "Text field_19" at 455,40 size 30x50; Text '9'
      Visibility <- "Digit_bl_10_THIS[1]_digarray[0]"
   Group "Group_1" at 455,40 size 38x50
   TextField "Text_dot_2" at 448,52 size 20x30; Text ','
      Visibility <- "Digit_bl_10_THIS{2}_visible0"
   TextField "Text field_20" at 430,40 size 30x50; Text '0'
      Visibility <- "Digit_bl_10_THIS[2]_digarray[0]"
   TextField "Text field_21" at 430,40 size 30x50; Text '1'
      Visibility <- "Digit_bl_10_THIS[2]_digarray[0]"
   TextField "Text field_22" at 430,40 size 30x50; Text '2'
      Visibility <- "Digit_bl_10_THIS[2]_digarray[0]"
   TextField "Text field_23" at 430,40 size 30x50; Text '3'
      Visibility <- "Digit_bl_10_THIS[2]_digarray[0]"
   TextField "Text field_24" at 430,40 size 30x50; Text '4'
      Visibility <- "Digit_bl_10_THIS[2]_digarray[0]"
   TextField "Text field_25" at 430,40 size 30x50; Text '5'
      Visibility <- "Digit_bl_10_THIS[2]_digarray[0]"
   TextField "Text field_26" at 430,40 size 30x50; Text '6'
      Visibility <- "Digit_bl_10_THIS[2]_digarray[0]"
   TextField "Text field_27" at 430,40 size 30x50; Text '7'
      Visibility <- "Digit_bl_10_THIS[2]_digarray[0]"
   TextField "Text field_28" at 430,40 size 30x50; Text '8'
      Visibility <- "Digit_bl_10_THIS[2]_digarray[0]"
   TextField "Text field_29" at 430,40 size 30x50; Text '9'
      Visibility <- "Digit_bl_10_THIS[2]_digarray[0]"
   Group "Group_2" at 430,40 size 38x50
   TextField "Text_dot_3" at 423,52 size 20x30; Text ','
      Visibility <- "Digit_bl_10_THIS{3}_visible0"
   TextField "Text field_30" at 405,40 size 30x50; Text '0'
      Visibility <- "Digit_bl_10_THIS[3]_digarray[0]"
   TextField "Text field_31" at 405,40 size 30x50; Text '1'
      Visibility <- "Digit_bl_10_THIS[3]_digarray[0]"
   TextField "Text field_32" at 405,40 size 30x50; Text '2'
      Visibility <- "Digit_bl_10_THIS[3]_digarray[0]"
   TextField "Text field_33" at 405,40 size 30x50; Text '3'
      Visibility <- "Digit_bl_10_THIS[3]_digarray[0]"
   TextField "Text field_34" at 405,40 size 30x50; Text '4'
      Visibility <- "Digit_bl_10_THIS[3]_digarray[0]"
   TextField "Text field_35" at 405,40 size 30x50; Text '5'
      Visibility <- "Digit_bl_10_THIS[3]_digarray[0]"
   TextField "Text field_36" at 405,40 size 30x50; Text '6'
      Visibility <- "Digit_bl_10_THIS[3]_digarray[0]"
   TextField "Text field_37" at 405,40 size 30x50; Text '7'
      Visibility <- "Digit_bl_10_THIS[3]_digarray[0]"
   TextField "Text field_38" at 405,40 size 30x50; Text '8'
      Visibility <- "Digit_bl_10_THIS[3]_digarray[0]"
   TextField "Text field_39" at 405,40 size 30x50; Text '9'
      Visibility <- "Digit_bl_10_THIS[3]_digarray[0]"
   Group "Group_3" at 405,40 size 38x50
   TextField "Text_dot_4" at 398,52 size 20x30; Text ','
      Visibility <- "Digit_bl_10_THIS{4}_visible0"
   TextField "Text field_40" at 380,40 size 30x50; Text '0'
      Visibility <- "Digit_bl_10_THIS[4]_digarray[0]"
   TextField "Text field_41" at 380,40 size 30x50; Text '1'
      Visibility <- "Digit_bl_10_THIS[4]_digarray[0]"
   TextField "Text field_42" at 380,40 size 30x50; Text '2'
      Visibility <- "Digit_bl_10_THIS[4]_digarray[0]"
   TextField "Text field_43" at 380,40 size 30x50; Text '3'
      Visibility <- "Digit_bl_10_THIS[4]_digarray[0]"
   TextField "Text field_44" at 380,40 size 30x50; Text '4'
      Visibility <- "Digit_bl_10_THIS[4]_digarray[0]"
   TextField "Text field_45" at 380,40 size 30x50; Text '5'
      Visibility <- "Digit_bl_10_THIS[4]_digarray[0]"
   TextField "Text field_46" at 380,40 size 30x50; Text '6'
      Visibility <- "Digit_bl_10_THIS[4]_digarray[0]"
   TextField "Text field_47" at 380,40 size 30x50; Text '7'
      Visibility <- "Digit_bl_10_THIS[4]_digarray[0]"
   TextField "Text field_48" at 380,40 size 30x50; Text '8'
      Visibility <- "Digit_bl_10_THIS[4]_digarray[0]"
   TextField "Text field_49" at 380,40 size 30x50; Text '9'
      Visibility <- "Digit_bl_10_THIS[4]_digarray[0]"
   Group "Group_4" at 380,40 size 38x50
   TextField "Text_dot_7" at 323,52 size 20x30; Text ','
      Visibility <- "Digit_bl_10_THIS{7}_visible0"
   TextField "Text field_70" at 305,40 size 30x50; Text '0'
      Visibility <- "Digit_bl_10_THIS[7]_digarray[0]"
   TextField "Text field_71" at 305,40 size 30x50; Text '1'
      Visibility <- "Digit_bl_10_THIS[7]_digarray[0]"
   TextField "Text field_72" at 305,40 size 30x50; Text '2'
      Visibility <- "Digit_bl_10_THIS[7]_digarray[0]"
   TextField "Text field_73" at 305,40 size 30x50; Text '3'
      Visibility <- "Digit_bl_10_THIS[7]_digarray[0]"
   TextField "Text field_74" at 305,40 size 30x50; Text '4'
      Visibility <- "Digit_bl_10_THIS[7]_digarray[0]"
   TextField "Text field_75" at 305,40 size 30x50; Text '5'
      Visibility <- "Digit_bl_10_THIS[7]_digarray[0]"
   TextField "Text field_76" at 305,40 size 30x50; Text '6'
      Visibility <- "Digit_bl_10_THIS[7]_digarray[0]"
   TextField "Text field_77" at 305,40 size 30x50; Text '7'
      Visibility <- "Digit_bl_10_THIS[7]_digarray[0]"
   TextField "Text field_78" at 305,40 size 30x50; Text '8'
      Visibility <- "Digit_bl_10_THIS[7]_digarray[0]"
   TextField "Text field_79" at 305,40 size 30x50; Text '9'
      Visibility <- "Digit_bl_10_THIS[7]_digarray[0]"
   Group "Group_7" at 305,40 size 38x50
   TextField "Text_dot_8" at 298,52 size 20x30; Text ','
      Visibility <- "Digit_bl_10_THIS{8}_visible0"
   TextField "Text field_80" at 280,40 size 30x50; Text '0'
      Visibility <- "Digit_bl_10_THIS[8]_digarray[0]"
   TextField "Text field_81" at 280,40 size 30x50; Text '1'
      Visibility <- "Digit_bl_10_THIS[8]_digarray[0]"
   TextField "Text field_82" at 280,40 size 30x50; Text '2'
      Visibility <- "Digit_bl_10_THIS[8]_digarray[0]"
   TextField "Text field_83" at 280,40 size 30x50; Text '3'
      Visibility <- "Digit_bl_10_THIS[8]_digarray[0]"
   TextField "Text field_84" at 280,40 size 30x50; Text '4'
      Visibility <- "Digit_bl_10_THIS[8]_digarray[0]"
   TextField "Text field_85" at 280,40 size 30x50; Text '5'
      Visibility <- "Digit_bl_10_THIS[8]_digarray[0]"
   TextField "Text field_86" at 280,40 size 30x50; Text '6'
      Visibility <- "Digit_bl_10_THIS[8]_digarray[0]"
   TextField "Text field_87" at 280,40 size 30x50; Text '7'
      Visibility <- "Digit_bl_10_THIS[8]_digarray[0]"
   TextField "Text field_88" at 280,40 size 30x50; Text '8'
      Visibility <- "Digit_bl_10_THIS[8]_digarray[0]"
   TextField "Text field_89" at 280,40 size 30x50; Text '9'
      Visibility <- "Digit_bl_10_THIS[8]_digarray[0]"
   Group "Group_8" at 280,40 size 38x50
   TextField "Text_dot_9" at 273,52 size 20x30; Text ','
      Visibility <- "Digit_bl_10_THIS{9}_visible0"
   TextField "Text field_90" at 255,40 size 30x50; Text '0'
      Visibility <- "Digit_bl_10_THIS[9]_digarray[0]"
   TextField "Text field_91" at 255,40 size 30x50; Text '1'
      Visibility <- "Digit_bl_10_THIS[9]_digarray[0]"
   TextField "Text field_92" at 255,40 size 30x50; Text '2'
      Visibility <- "Digit_bl_10_THIS[9]_digarray[0]"
   TextField "Text field_93" at 255,40 size 30x50; Text '3'
      Visibility <- "Digit_bl_10_THIS[9]_digarray[0]"
   TextField "Text field_94" at 255,40 size 30x50; Text '4'
      Visibility <- "Digit_bl_10_THIS[9]_digarray[0]"
   TextField "Text field_95" at 255,40 size 30x50; Text '5'
      Visibility <- "Digit_bl_10_THIS[9]_digarray[0]"
   TextField "Text field_96" at 255,40 size 30x50; Text '6'
      Visibility <- "Digit_bl_10_THIS[9]_digarray[0]"
   TextField "Text field_97" at 255,40 size 30x50; Text '7'
      Visibility <- "Digit_bl_10_THIS[9]_digarray[0]"
   TextField "Text field_98" at 255,40 size 30x50; Text '8'
      Visibility <- "Digit_bl_10_THIS[9]_digarray[0]"
   TextField "Text field_99" at 255,40 size 30x50; Text '9'
      Visibility <- "Digit_bl_10_THIS[9]_digarray[0]"
   Group "Group_9" at 255,40 size 38x50
   TextField "Text_dot_10" at 248,52 size 20x30; Text ','
      Visibility <- "Digit_bl_10_THIS{10}_visible0"
   TextField "Text field_100" at 230,40 size 30x50; Text '0'
      Visibility <- "Digit_bl_10_THIS[10]_digarray[0]"
   TextField "Text field_101" at 230,40 size 30x50; Text '1'
      Visibility <- "Digit_bl_10_THIS[10]_digarray[0]"
   TextField "Text field_102" at 230,40 size 30x50; Text '2'
      Visibility <- "Digit_bl_10_THIS[10]_digarray[0]"
   TextField "Text field_103" at 230,40 size 30x50; Text '3'
      Visibility <- "Digit_bl_10_THIS[10]_digarray[0]"
   TextField "Text field_104" at 230,40 size 30x50; Text '4'
      Visibility <- "Digit_bl_10_THIS[10]_digarray[0]"
   TextField "Text field_105" at 230,40 size 30x50; Text '5'
      Visibility <- "Digit_bl_10_THIS[10]_digarray[0]"
   TextField "Text field_106" at 230,40 size 30x50; Text '6'
      Visibility <- "Digit_bl_10_THIS[10]_digarray[0]"
   TextField "Text field_107" at 230,40 size 30x50; Text '7'
      Visibility <- "Digit_bl_10_THIS[10]_digarray[0]"
   TextField "Text field_108" at 230,40 size 30x50; Text '8'
      Visibility <- "Digit_bl_10_THIS[10]_digarray[0]"
   TextField "Text field_109" at 230,40 size 30x50; Text '9'
      Visibility <- "Digit_bl_10_THIS[10]_digarray[0]"
   Group "Group_10" at 230,40 size 38x50
   TextField "Text_dot_13" at 173,52 size 20x30; Text ','
      Visibility <- "Digit_bl_10_THIS{13}_visible0"
   TextField "Text field_130" at 155,40 size 30x50; Text '0'
      Visibility <- "Digit_bl_10_THIS[13]_digarray[0]"
   TextField "Text field_131" at 155,40 size 30x50; Text '1'
      Visibility <- "Digit_bl_10_THIS[13]_digarray[0]"
   TextField "Text field_132" at 155,40 size 30x50; Text '2'
      Visibility <- "Digit_bl_10_THIS[13]_digarray[0]"
   TextField "Text field_133" at 155,40 size 30x50; Text '3'
      Visibility <- "Digit_bl_10_THIS[13]_digarray[0]"
   TextField "Text field_134" at 155,40 size 30x50; Text '4'
      Visibility <- "Digit_bl_10_THIS[13]_digarray[0]"
   TextField "Text field_135" at 155,40 size 30x50; Text '5'
      Visibility <- "Digit_bl_10_THIS[13]_digarray[0]"
   TextField "Text field_136" at 155,40 size 30x50; Text '6'
      Visibility <- "Digit_bl_10_THIS[13]_digarray[0]"
   TextField "Text field_137" at 155,40 size 30x50; Text '7'
      Visibility <- "Digit_bl_10_THIS[13]_digarray[0]"
   TextField "Text field_138" at 155,40 size 30x50; Text '8'
      Visibility <- "Digit_bl_10_THIS[13]_digarray[0]"
   TextField "Text field_139" at 155,40 size 30x50; Text '9'
      Visibility <- "Digit_bl_10_THIS[13]_digarray[0]"
   Group "Group_13" at 155,40 size 38x50
   TextField "Text_dot_14" at 148,52 size 20x30; Text ','
      Visibility <- "Digit_bl_10_THIS{14}_visible0"
   TextField "Text field_140" at 130,40 size 30x50; Text '0'
      Visibility <- "Digit_bl_10_THIS[14]_digarray[0]"
   TextField "Text field_141" at 130,40 size 30x50; Text '1'
      Visibility <- "Digit_bl_10_THIS[14]_digarray[0]"
   TextField "Text field_142" at 130,40 size 30x50; Text '2'
      Visibility <- "Digit_bl_10_THIS[14]_digarray[0]"
   TextField "Text field_143" at 130,40 size 30x50; Text '3'
      Visibility <- "Digit_bl_10_THIS[14]_digarray[0]"
   TextField "Text field_144" at 130,40 size 30x50; Text '4'
      Visibility <- "Digit_bl_10_THIS[14]_digarray[0]"
   TextField "Text field_145" at 130,40 size 30x50; Text '5'
      Visibility <- "Digit_bl_10_THIS[14]_digarray[0]"
   TextField "Text field_146" at 130,40 size 30x50; Text '6'
      Visibility <- "Digit_bl_10_THIS[14]_digarray[0]"
   TextField "Text field_147" at 130,40 size 30x50; Text '7'
      Visibility <- "Digit_bl_10_THIS[14]_digarray[0]"
   TextField "Text field_148" at 130,40 size 30x50; Text '8'
      Visibility <- "Digit_bl_10_THIS[14]_digarray[0]"
   TextField "Text field_149" at 130,40 size 30x50; Text '9'
      Visibility <- "Digit_bl_10_THIS[14]_digarray[0]"
   Group "Group_14" at 130,40 size 38x50
   TextField "Text_dot_15" at 123,52 size 20x30; Text ','
      Visibility <- "Digit_bl_10_THIS{15}_visible0"
   TextField "Text field_150" at 105,40 size 30x50; Text '0'
      Visibility <- "Digit_bl_10_THIS[15]_digarray[0]"
   TextField "Text field_151" at 105,40 size 30x50; Text '1'
      Visibility <- "Digit_bl_10_THIS[15]_digarray[0]"
   TextField "Text field_152" at 105,40 size 30x50; Text '2'
      Visibility <- "Digit_bl_10_THIS[15]_digarray[0]"
   TextField "Text field_153" at 105,40 size 30x50; Text '3'
      Visibility <- "Digit_bl_10_THIS[15]_digarray[0]"
   TextField "Text field_154" at 105,40 size 30x50; Text '4'
      Visibility <- "Digit_bl_10_THIS[15]_digarray[0]"
   TextField "Text field_155" at 105,40 size 30x50; Text '5'
      Visibility <- "Digit_bl_10_THIS[15]_digarray[0]"
   TextField "Text field_156" at 105,40 size 30x50; Text '6'
      Visibility <- "Digit_bl_10_THIS[15]_digarray[0]"
   TextField "Text field_157" at 105,40 size 30x50; Text '7'
      Visibility <- "Digit_bl_10_THIS[15]_digarray[0]"
   TextField "Text field_158" at 105,40 size 30x50; Text '8'
      Visibility <- "Digit_bl_10_THIS[15]_digarray[0]"
   TextField "Text field_159" at 105,40 size 30x50; Text '9'
      Visibility <- "Digit_bl_10_THIS[15]_digarray[0]"
   Group "Group_15" at 105,40 size 38x50
   TextField "Text_dot_5" at 373,52 size 20x30; Text ','
      Visibility <- "Digit_bl_10_THIS{5}_visible0"
   TextField "Text field_50" at 355,40 size 30x50; Text '0'
      Visibility <- "Digit_bl_10_THIS[5]_digarray[0]"
   TextField "Text field_51" at 355,40 size 30x50; Text '1'
      Visibility <- "Digit_bl_10_THIS[5]_digarray[0]"
   TextField "Text field_52" at 355,40 size 30x50; Text '2'
      Visibility <- "Digit_bl_10_THIS[5]_digarray[0]"
   TextField "Text field_53" at 355,40 size 30x50; Text '3'
      Visibility <- "Digit_bl_10_THIS[5]_digarray[0]"
   TextField "Text field_54" at 355,40 size 30x50; Text '4'
      Visibility <- "Digit_bl_10_THIS[5]_digarray[0]"
   TextField "Text field_55" at 355,40 size 30x50; Text '5'
      Visibility <- "Digit_bl_10_THIS[5]_digarray[0]"
   TextField "Text field_56" at 355,40 size 30x50; Text '6'
      Visibility <- "Digit_bl_10_THIS[5]_digarray[0]"
   TextField "Text field_57" at 355,40 size 30x50; Text '7'
      Visibility <- "Digit_bl_10_THIS[5]_digarray[0]"
   TextField "Text field_58" at 355,40 size 30x50; Text '8'
      Visibility <- "Digit_bl_10_THIS[5]_digarray[0]"
   TextField "Text field_59" at 355,40 size 30x50; Text '9'
      Visibility <- "Digit_bl_10_THIS[5]_digarray[0]"
   Group "Group_5" at 355,40 size 38x50
   TextField "Text_dot_6" at 348,52 size 20x30; Text ','
      Visibility <- "Digit_bl_10_THIS{6}_visible0"
   TextField "Text field_60" at 330,40 size 30x50; Text '0'
      Visibility <- "Digit_bl_10_THIS[6]_digarray[0]"
   TextField "Text field_61" at 330,40 size 30x50; Text '1'
      Visibility <- "Digit_bl_10_THIS[6]_digarray[0]"
   TextField "Text field_62" at 330,40 size 30x50; Text '2'
      Visibility <- "Digit_bl_10_THIS[6]_digarray[0]"
   TextField "Text field_63" at 330,40 size 30x50; Text '3'
      Visibility <- "Digit_bl_10_THIS[6]_digarray[0]"
   TextField "Text field_64" at 330,40 size 30x50; Text '4'
      Visibility <- "Digit_bl_10_THIS[6]_digarray[0]"
   TextField "Text field_65" at 330,40 size 30x50; Text '5'
      Visibility <- "Digit_bl_10_THIS[6]_digarray[0]"
   TextField "Text field_66" at 330,40 size 30x50; Text '6'
      Visibility <- "Digit_bl_10_THIS[6]_digarray[0]"
   TextField "Text field_67" at 330,40 size 30x50; Text '7'
      Visibility <- "Digit_bl_10_THIS[6]_digarray[0]"
   TextField "Text field_68" at 330,40 size 30x50; Text '8'
      Visibility <- "Digit_bl_10_THIS[6]_digarray[0]"
   TextField "Text field_69" at 330,40 size 30x50; Text '9'
      Visibility <- "Digit_bl_10_THIS[6]_digarray[0]"
   Group "Group_6" at 330,40 size 38x50
   TextField "Text_dot_11" at 223,52 size 20x30; Text ','
      Visibility <- "Digit_bl_10_THIS{11}_visible0"
   TextField "Text field_110" at 205,40 size 30x50; Text '0'
      Visibility <- "Digit_bl_10_THIS[11]_digarray[0]"
   TextField "Text field_111" at 205,40 size 30x50; Text '1'
      Visibility <- "Digit_bl_10_THIS[11]_digarray[0]"
   TextField "Text field_112" at 205,40 size 30x50; Text '2'
      Visibility <- "Digit_bl_10_THIS[11]_digarray[0]"
   TextField "Text field_113" at 205,40 size 30x50; Text '3'
      Visibility <- "Digit_bl_10_THIS[11]_digarray[0]"
   TextField "Text field_114" at 205,40 size 30x50; Text '4'
      Visibility <- "Digit_bl_10_THIS[11]_digarray[0]"
   TextField "Text field_115" at 205,40 size 30x50; Text '5'
      Visibility <- "Digit_bl_10_THIS[11]_digarray[0]"
   TextField "Text field_116" at 205,40 size 30x50; Text '6'
      Visibility <- "Digit_bl_10_THIS[11]_digarray[0]"
   TextField "Text field_117" at 205,40 size 30x50; Text '7'
      Visibility <- "Digit_bl_10_THIS[11]_digarray[0]"
   TextField "Text field_118" at 205,40 size 30x50; Text '8'
      Visibility <- "Digit_bl_10_THIS[11]_digarray[0]"
   TextField "Text field_119" at 205,40 size 30x50; Text '9'
      Visibility <- "Digit_bl_10_THIS[11]_digarray[0]"
   Group "Group_11" at 205,40 size 38x50
   TextField "Text_dot_12" at 198,52 size 20x30; Text ','
      Visibility <- "Digit_bl_10_THIS{12}_visible0"
   TextField "Text field_120" at 180,40 size 30x50; Text '0'
      Visibility <- "Digit_bl_10_THIS[12]_digarray[0]"
   TextField "Text field_121" at 180,40 size 30x50; Text '1'
      Visibility <- "Digit_bl_10_THIS[12]_digarray[0]"
   TextField "Text field_122" at 180,40 size 30x50; Text '2'
      Visibility <- "Digit_bl_10_THIS[12]_digarray[0]"
   TextField "Text field_123" at 180,40 size 30x50; Text '3'
      Visibility <- "Digit_bl_10_THIS[12]_digarray[0]"
   TextField "Text field_124" at 180,40 size 30x50; Text '4'
      Visibility <- "Digit_bl_10_THIS[12]_digarray[0]"
   TextField "Text field_125" at 180,40 size 30x50; Text '5'
      Visibility <- "Digit_bl_10_THIS[12]_digarray[0]"
   TextField "Text field_126" at 180,40 size 30x50; Text '6'
      Visibility <- "Digit_bl_10_THIS[12]_digarray[0]"
   TextField "Text field_127" at 180,40 size 30x50; Text '7'
      Visibility <- "Digit_bl_10_THIS[12]_digarray[0]"
   TextField "Text field_128" at 180,40 size 30x50; Text '8'
      Visibility <- "Digit_bl_10_THIS[12]_digarray[0]"
   TextField "Text field_129" at 180,40 size 30x50; Text '9'
      Visibility <- "Digit_bl_10_THIS[12]_digarray[0]"
   Group "Group_12" at 180,40 size 38x50
   TextField "Text field_160" at 280,45 size 225x40; Text 'E r r o r'
      Visibility <- "NUMs_Error"
   Group "Group" at 85,55 size 400x10
   TextField "Text minus_15" at 85,55 size 25x10; Text '_'
      Visibility <- "Digit_bl_10_THIS{15}_visiMinus"
   TextField "Text minus_1" at 435,55 size 25x10; Text '_'
      Visibility <- "Digit_bl_10_THIS{1}_visiMinus"
   TextField "Text minus_2" at 410,55 size 25x10; Text '_'
      Visibility <- "Digit_bl_10_THIS{2}_visiMinus"
   TextField "Text minus_3" at 385,55 size 25x10; Text '_'
      Visibility <- "Digit_bl_10_THIS{3}_visiMinus"
   TextField "Text minus_4" at 360,55 size 25x10; Text '_'
      Visibility <- "Digit_bl_10_THIS{4}_visiMinus"
   TextField "Text minus_5" at 335,55 size 25x10; Text '_'
      Visibility <- "Digit_bl_10_THIS{5}_visiMinus"
   TextField "Text minus_6" at 310,55 size 25x10; Text '_'
      Visibility <- "Digit_bl_10_THIS{6}_visiMinus"
   TextField "Text minus_7" at 285,55 size 25x10; Text '_'
      Visibility <- "Digit_bl_10_THIS{7}_visiMinus"
   TextField "Text minus_8" at 260,55 size 25x10; Text '_'
      Visibility <- "Digit_bl_10_THIS{8}_visiMinus"
   TextField "Text minus_9" at 235,55 size 25x10; Text '_'
      Visibility <- "Digit_bl_10_THIS{9}_visiMinus"
   TextField "Text minus_10" at 210,55 size 25x10; Text '_'
      Visibility <- "Digit_bl_10_THIS{10}_visiMinus"
   TextField "Text minus_11" at 185,55 size 25x10; Text '_'
      Visibility <- "Digit_bl_10_THIS{11}_visiMinus"
   TextField "Text minus_12" at 160,55 size 25x10; Text '_'
      Visibility <- "Digit_bl_10_THIS{12}_visiMinus"
   TextField "Text minus_13" at 135,55 size 25x10; Text '_'
      Visibility <- "Digit_bl_10_THIS{13}_visiMinus"
   TextField "Text minus_14" at 110,55 size 25x10; Text '_'
      Visibility <- "Digit_bl_10_THIS{14}_visiMinus"
   TextField "Text minus_0" at 460,55 size 25x10; Text '_'
      Visibility <- "Digit_bl_10_THIS{0}_visiMinus"

Template "Template_1" 800x420
   Button "Exit" at 720,360 size 78x58; TextOff 'Exit'; PictureOff "ExitRuntime_TP900_Comfort_TR"; PictureOn "ExitRuntime_TP900_Comfort_TR"
      on Release: StopRuntime(0)
   Button "Template_Button" at 640,360 size 78x58; TextOff 'Text'
   Button "Template_Button_1" at 560,360 size 78x58; TextOff 'Text'
   Button "Template_Button_2" at 480,360 size 78x58; TextOff 'Text'
   Button "Template_Button_3" at 400,360 size 78x58; TextOff 'Text'
   Button "Template_Button_4" at 321,360 size 78x58; TextOff 'Text'
   Button "Template_Button_5" at 241,360 size 78x58; TextOff 'Text'
   Button "Template_Button_6" at 161,360 size 78x58; TextOff 'Text'
   Button "Template_Button_7" at 81,360 size 78x58; TextOff 'Text'
   Button "Start screen" at 1,360 size 78x58; TextOff 'Start screen'; PictureOff "NavigateHome_TP900_Comfort_TR"; PictureOn "NavigateHome_TP900_Comfort_TR"
      on Release: ActivateScreen("Root screen", 0)
*)